PROGRAM MAIN
VAR
END_VAR

PI_CNTRL_SIM_CLOSED_LOOP();

END_PROGRAM

(* stored: Version 1.1.0.1, ProductVersion 3.1.4024.9
   POU MAIN: Id {d2280aa5-b837-4d67-9302-e0ce9032e37d}, SpecialFunc None *)
